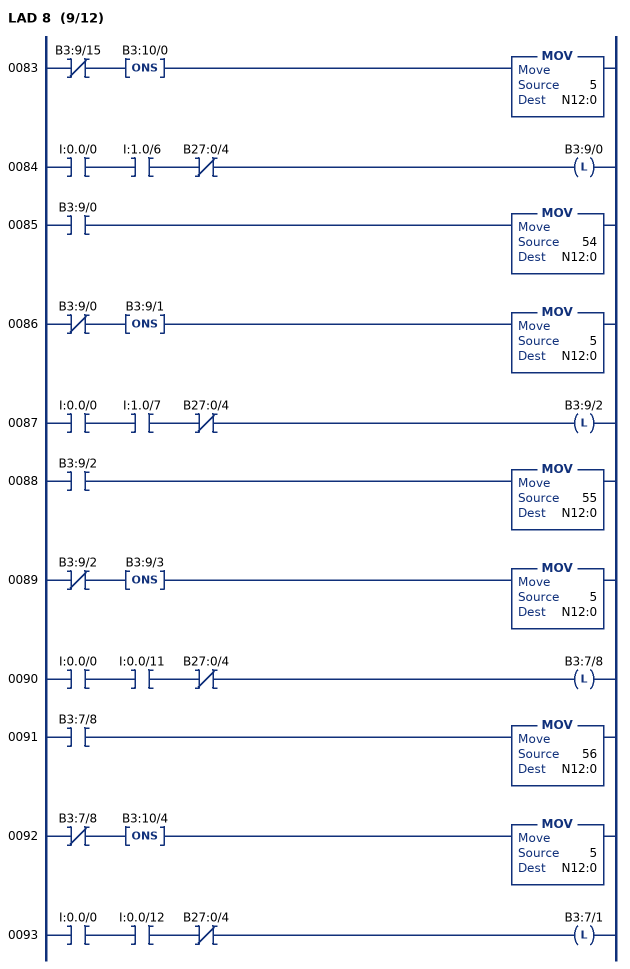
% Rung: 83 %
SOR XIO B3:9/15 ONS B3:10/0 MOV 5 N12:0 EOR
% Rung: 84 %
SOR XIC I:0.0/0 XIC I:1.0/6 XIO B27:0/4 OTL B3:9/0 EOR
% Rung: 85 %
SOR XIC B3:9/0 MOV 54 N12:0 EOR
% Rung: 86 %
SOR XIO B3:9/0 ONS B3:9/1 MOV 5 N12:0 EOR
% Rung: 87 %
SOR XIC I:0.0/0 XIC I:1.0/7 XIO B27:0/4 OTL B3:9/2 EOR
% Rung: 88 %
SOR XIC B3:9/2 MOV 55 N12:0 EOR
% Rung: 89 %
SOR XIO B3:9/2 ONS B3:9/3 MOV 5 N12:0 EOR
% Rung: 90 %
SOR XIC I:0.0/0 XIC I:0.0/11 XIO B27:0/4 OTL B3:7/8 EOR
% Rung: 91 %
SOR XIC B3:7/8 MOV 56 N12:0 EOR
% Rung: 92 %
SOR XIO B3:7/8 ONS B3:10/4 MOV 5 N12:0 EOR
% Rung: 93 %
SOR XIC I:0.0/0 XIC I:0.0/12 XIO B27:0/4 OTL B3:7/1 EOR

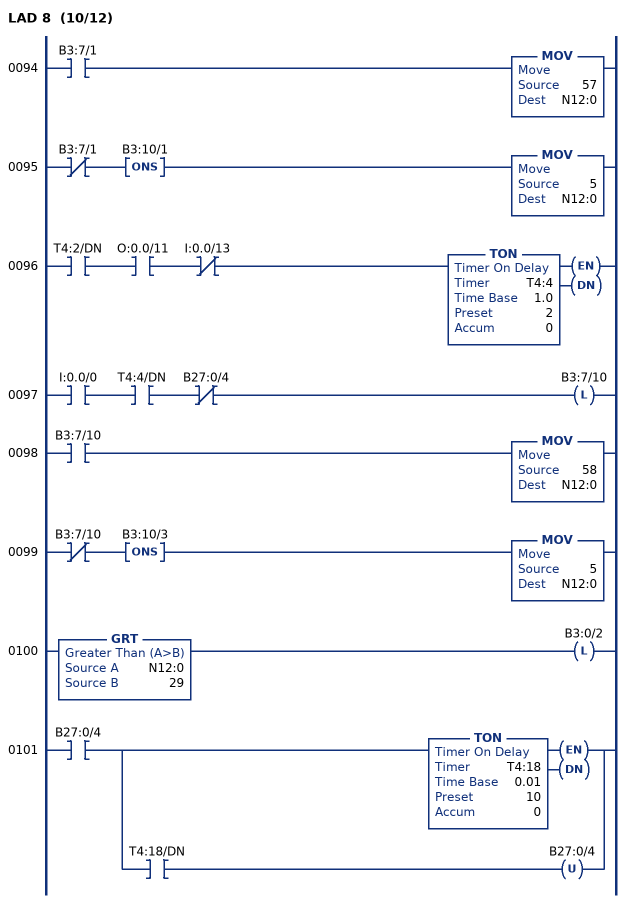
% Rung: 94 %
SOR XIC B3:7/1 MOV 57 N12:0 EOR
% Rung: 95 %
SOR XIO B3:7/1 ONS B3:10/1 MOV 5 N12:0 EOR
% Rung: 96 %
SOR XIC T4:2/DN XIC O:0.0/11 XIO I:0.0/13 TON T4:4 1.0 2 0 EOR
% Rung: 97 %
SOR XIC I:0.0/0 XIC T4:4/DN XIO B27:0/4 OTL B3:7/10 EOR
% Rung: 98 %
SOR XIC B3:7/10 MOV 58 N12:0 EOR
% Rung: 99 %
SOR XIO B3:7/10 ONS B3:10/3 MOV 5 N12:0 EOR
% Rung: 100 %
SOR GRT N12:0 29 OTL B3:0/2 EOR
% Rung: 101 %
SOR XIC B27:0/4 BST TON T4:18 0.01 10 0 NXB XIC T4:18/DN OTU B27:0/4 BND EOR

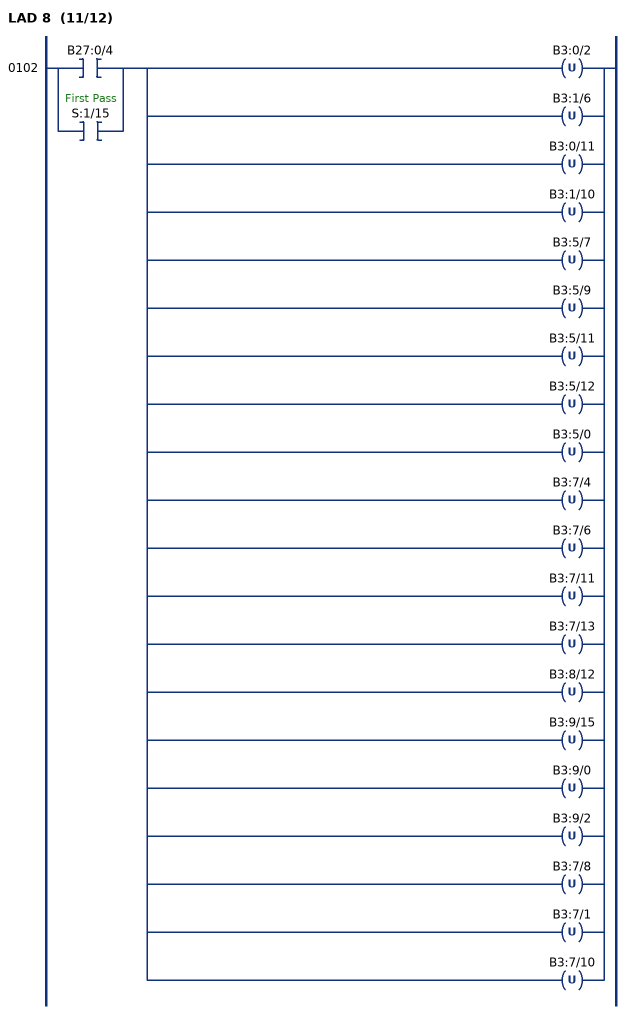
% Rung: 102 %
SOR BST XIC B27:0/4 NXB XIC S:1/15 BND BST OTU B3:0/2 NXB OTU B3:1/6 NXB OTU B3:0/11 NXB OTU B3:1/10 NXB OTU B3:5/7 NXB OTU B3:5/9 NXB OTU B3:5/11 NXB OTU B3:5/12 NXB OTU B3:5/0 NXB OTU B3:7/4 NXB OTU B3:7/6 NXB OTU B3:7/11 NXB OTU B3:7/13 NXB OTU B3:8/12 NXB OTU B3:9/15 NXB OTU B3:9/0 NXB OTU B3:9/2 NXB OTU B3:7/8 NXB OTU B3:7/1 NXB OTU B3:7/10 BND EOR
%   S:1/15  "First Pass" %

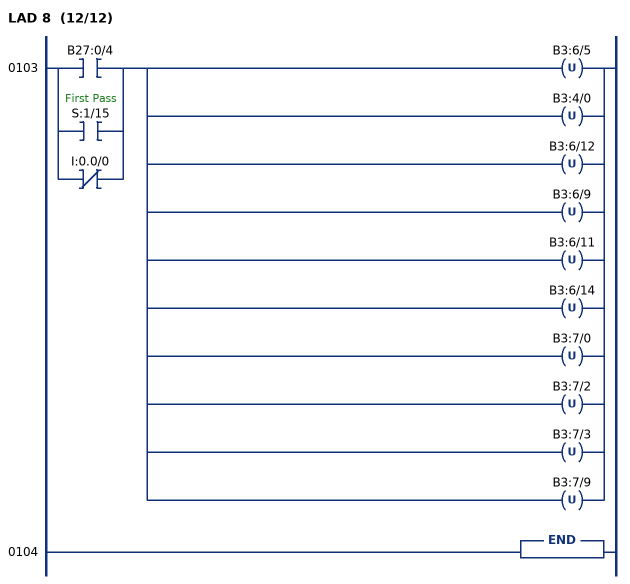
% Rung: 103 %
SOR BST XIC B27:0/4 NXB XIC S:1/15 NXB XIO I:0.0/0 BND BST OTU B3:6/5 NXB OTU B3:4/0 NXB OTU B3:6/12 NXB OTU B3:6/9 NXB OTU B3:6/11 NXB OTU B3:6/14 NXB OTU B3:7/0 NXB OTU B3:7/2 NXB OTU B3:7/3 NXB OTU B3:7/9 BND EOR
%   S:1/15  "First Pass" %
% Rung: 104 %
SOR END EOR

DATA TABLE (non-zero values as saved)
DATA B3
% B3:0 % 0X2010 0X4084 0X0229 0X1424 0X554C 0XC120 0X0410 0X10A0 0XEB9D 0X77CA
% B3:10 % 0X003F 0X0000 0X0000 0X0000 0X0000 0X0000 0X0000 0X0000 0X0000 0X0000
DATA T4
% .PRE .ACC %
% T4:2 % 800 800
% T4:3 % 100 0
% T4:4 % 2 0
% T4:5 % 10 10
% T4:6 % 100 0
% T4:7 % 50 0
% T4:8 % 4 4
% T4:13 % 100 0
% T4:15 % 4 4
% T4:18 % 10 0
DATA N7
% N7:0 % 9 0 0 0 0 0 0 0 0 0
DATA N10
% N10:0 % 200 350 700 170 250 430 850 320 500 750
DATA N12
% N12:0 % 5 2
DATA N13
% N13:0 % 525 525 525 525 525 525 525 525 525 525
DATA N17
% N17:0 % 28
DATA ST23
% ST23:0 % "tj,s green dressing"
% ST23:1 % "250 ML"
% ST23:2 % "400 ML"
% ST23:3 % "11.75 oz"
% ST23:4 % "354 ML"
% ST23:5 % "450 ML"
% ST23:6 % "TBD"
% ST23:7 % "tj,s green dressing"
% ST23:8 % "16 OZ"
% ST23:9 % "tj,s green dressing"
% ST23:10 % "tj,s green dressing"
% ST23:11 % "tj,s green dressing"
% ST23:12 % "11 oz round"
% ST23:31 % "tj,s green dressing"
